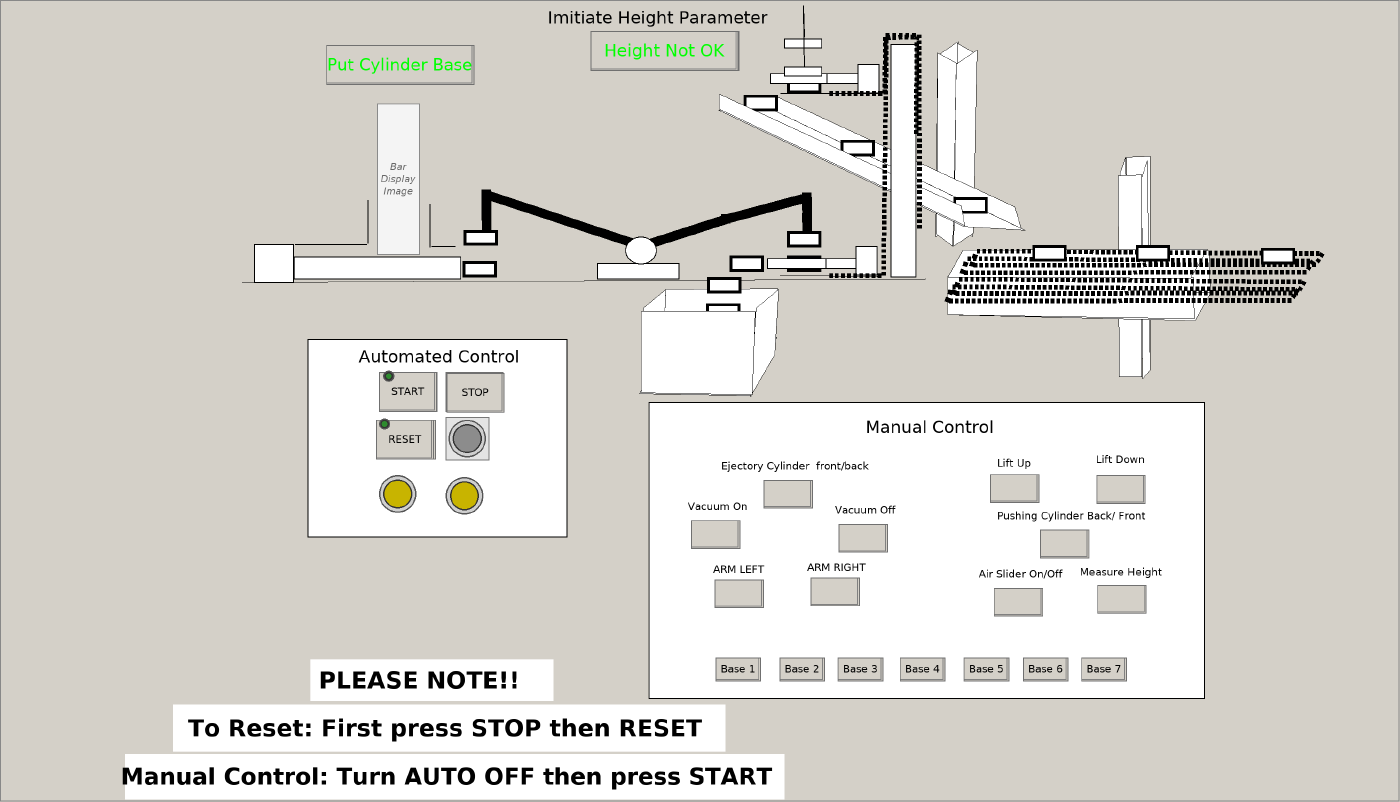
VISUALIZATION StationVisual  // 1489x854
    RoundedRectangle (837,272 36x17), invisible if: StationVisualProgram.MagPos5
    RoundedRectangle (816,275 105x11), invisible if: StationVisualProgram.EjecCylDown
    RoundedRectangle (837,82 36x17), invisible if: StationVisualProgram.BasePos6
    RoundedRectangle (819,78 105x11), invisible if: StationVisualProgram.EjecCylUp
    Polygon (684,328) (708,308) (706,360) (684,419)
    Polygon (708,308) (827,307) (824,362) (706,360)
    Polygon (707,359) (826,359) (798,421) (680,419)
    Polygon (804,328) (828,308) (824,377) (798,422)
    RoundedRectangle (751,323 36x17), invisible if: StationVisualProgram.BasePos8b
    Group (995,44 44x297)
        Polygon (0,208) (2,15) (24,0) (20,195)
        Polygon (22,195) (23,2) (43,13) (39,208)
        Polygon (19,218) (22,24) (44,9) (40,204)
        Polygon (1,205) (2,12) (22,23) (18,218)
    Polygon (764,117) (1025,241) (1090,245) (824,118)
    Polygon (822,117) (1086,243) (1079,220) (822,101)
    Group (1189,166 50x236)
        Polygon (3,233) (2,19) (8,1) (11,224)
        Polygon (10,215) (9,1) (34,0) (34,215)
        Polygon (1,235) (0,21) (25,20) (25,235)
        Polygon (26,237) (25,23) (31,5) (34,228)
    Polyline (680,261) (517,207) (517,217) (517,225) (517,230) (517,246), invisible if: Arm_put
    Polyline (685,261) (772,233) (858,210) (858,219) (858,232) (858,246), invisible if: Arm_take
    Rectangle (401,138 43x121), invisible if: RotDriveMag
    Line (391,229)
    Line (391,213) (391,259)
    Line (457,217) (457,263)
    Line (314,260) (390,260)
    Line (984,297) (258,301)
    Line (459,262) (484,262)
    Rectangle (287,273 106x24), invisible if: Mag_front
    RoundedRectangle (404,276 36x17), invisible if: StationVisualProgram.MagPos1
    RoundedRectangle (492,278 36x17), invisible if: StationVisualProgram.MagPos2
    BarDisplayImage (401,110 45x161), value: DistStationSensors.Current, style: BarDisplayImage-Gray, scale format: %.1f, scale 0..8
    Button (347,48 157x42), "Put Cylinder Base"
        tap insertMag
    Group (635,252 87x45)
        RoundedRectangle (0,28 87x17)
        Ellipse (30,0 33x29)
    RoundedRectangle (837,246 36x17), invisible if: StationVisualProgram.MagPos4
    RoundedRectangle (493,245 36x16), invisible if: StationVisualProgram.MagPos3
    Group (327,361 278x211)
        Rectangle (0,0 276x211)
        Group (147,35 50x28)
            Button (0,0 61x42), "STOP"
                toggle stop
            Button (1,1 61x42), "STOP", invisible if: stop
                toggle stop
        PushSwitchLed (142,83 56x46), tooltip "AUTO/Manual", variable: Automan, behaviour: TOGGLE, style: Switch-PushSwitchLed-Gray
        Lamp1 (68,142 56x46), tooltip "Indicaotor 1", variable: Mat_sen, style: Lamp-Lamp1-Yellow
        Lamp1 (139,144 56x46), tooltip "Indicator 2", style: Lamp-Lamp1-Yellow
        Label (2,7 276x24), "Automated Control"
        Group (76,35 50x28)
            Button (1,0 61x42), "START"
                toggle start
            Button (0,0 61x42), "START", invisible if: start
                toggle start
        Group (73,86 51x28)
            Button (2,0 61x42), "RESET"
                toggle reset
            Button (0,0 61x42), "RESET", invisible if: reset
                toggle reset
        Lamp1 (75,33 23x13), variable: L_START, style: Lamp-Lamp1-Green
        Lamp1 (72,84 20x13), variable: L_RESET, style: Lamp-Lamp1-Green
    Group (1008,265 479x76)
        Polygon (263,76) (1,70) (20,20) (281,44)
        Polygon (279,46) (17,42) (17,1) (278,2)
        Polygon (262,74) (0,70) (0,29) (261,30)
        Polygon (258,31) (0,30) (16,1) (276,0)
    Group (1007,267 476x30)
        Polyline (6,38) (373,41) (366,53) (0,54) (6,38)
        Polyline (13,30) (380,33) (373,45) (7,46) (13,30)
        Polyline (22,8) (389,11) (382,23) (16,24) (22,8)
        Polyline (32,0) (399,3) (392,15) (26,16) (32,0)
    RoundedRectangle (791,101 36x17), invisible if: StationVisualProgram.BasePos7
    RoundedRectangle (1098,261 36x17), invisible if: StationVisualProgram.BasePos7c
    RoundedRectangle (1208,261 36x17), invisible if: StationVisualProgram.BasePos7d
    RoundedRectangle (1341,264 36x17), invisible if: StationVisualProgram.BasePos7e
    RoundedRectangle (776,272 36x17), invisible if: StationVisualProgram.BasePos8
    RoundedRectangle (894,149 36x17), invisible if: StationVisualProgram.BasePos7a
    RoundedRectangle (1014,210 36x17), invisible if: StationVisualProgram.BasePos7b
    Group (878,262 55x31), invisible if: Lift_Up
        RoundedRectangle (0,13 50x11)
        RoundedRectangle (32,0 23x31)
    Group (879,68 56x31), invisible if: Lift_Down
        RoundedRectangle (0,10 50x11), invisible if: Lift_Down
        RoundedRectangle (33,0 23x31), invisible if: Lift_Down
    RoundedRectangle (752,295 36x17), invisible if: StationVisualProgram.BasePos8a
    Polygon (682,331) (803,331) (800,420) (682,418)
    Group (834,6 40x45), invisible if: H_Meas
        RoundedRectangle (0,35 40x10)
        Line (20,0) (21,33)
    Group (834,9 40x72), invisible if: StationVisualProgram.H_MeasCylDo
        Line (20,0) (21,66)
        RoundedRectangle (0,62 40x10)
    Rectangle (313,273 177x24), invisible if: Mag_back
    RoundedRectangle (270,260 42x41)
    Button (629,33 157x42), "Height OK"
        toggle Work_ok
    Button (628,33 157x42), "Height Not OK", invisible if: Work_ok
        toggle Work_ok
    Label (579,4 241x30), "Imitiate Height Parameter"
    Polygon (765,116) (1026,240) (1022,219) (765,100)
    RoundedRectangle (947,47 27x248)
    Group (830,39 145x255), invisible if: Lift_Up
        Polyline (52,254) (110,254) (113,1) (145,0) (144,106)
        Line (0,254) (103,255)
    Group (830,37 148x209), invisible if: Lift_Down
        Polyline (52,62) (111,62) (112,0) (147,0) (148,209)
        Line (0,62) (105,62)
    Rectangle (690,428 591x316)
    Label (851,443 276x24), "Manual Control"
    Group (676,509 175x75)
        Button (59,45 52x30)
            tap Vacumon
        Label (0,0 175x61), "Vacuum On"
    Group (698,576 175x71)
        Button (62,41 52x30)
            tap Armleft
        Label (0,0 175x61), "ARM LEFT"
    Group (802,574 175x71)
        Button (60,41 52x30)
            tap Armright
        Label (0,0 175x61), "ARM RIGHT"
    Group (758,466 175x75)
        Label (0,0 175x61), "Ejectory Cylinder front/back"
        Button (54,45 52x30), colour toggle: Mag
            toggle Mag
    Group (833,513 175x75)
        Button (59,45 52x30)
            tap Vacumoff
        Label (0,0 175x61), "Vacuum Off"
    Group (998,581 175x75)
        Button (59,45 52x30), colour toggle: Slide
            toggle Slide
        Label (0,0 175x61), "Air Slider On/Off"
    Group (991,463 175x72)
        Button (62,42 52x30)
            tap LiftUp
        Label (0,0 175x61), "Lift Up"
    Group (1104,459 175x77)
        Button (62,47 52x30)
            tap LiftDown
        Label (0,0 175x61), "Lift Down"
    Group (1052,519 175x75)
        Label (0,0 175x61), "Pushing Cylinder Back/ Front"
        Button (54,45 52x30)
            toggle MatPush
    Button (1167,623 52x30)
        toggle H_Meas
    Label (1105,579 175x61), "Measure Height"
    Button (761,700 48x25), "Base 1"
        toggle StationVisualProgram.MagPos1
    Button (829,700 48x25), "Base 2"
        toggle StationVisualProgram.MagPos2
    Button (891,700 48x25), "Base 3"
        toggle StationVisualProgram.MagPos3
    Button (957,700 48x25), "Base 4"
        toggle StationVisualProgram.MagPos4
    Button (1025,700 48x25), "Base 5"
        toggle StationVisualProgram.MagPos5
    Button (1088,700 48x25), "Base 6"
        toggle StationVisualProgram.BasePos6
    Button (1150,700 48x25), "Base 7"
        toggle StationVisualProgram.BasePos7
    Label (610,359 268x30), "REJECTED :("
    Group (132,701 703x151)
        Textfield (197,0 260x46), "PLEASE NOTE!!"
        Textfield (51,48 589x52), "To Reset: First press STOP then RESET"
        Textfield (0,101 703x50), "Manual Control: Turn AUTO OFF then press START"
END_VISUALIZATION

(* stored: Version 1.1.0.1, ProductVersion 3.1.4018.5
   Visu StationVisual: Id {20fed742-46c6-4b30-bb76-324332019ff6} *)
